FUNCTION_BLOCK FB_Transport_A
VAR_INPUT
	bStop1 :BOOL;
	bStop2 :BOOL;
	bStop3 :BOOL;
END_VAR
VAR_OUTPUT
	//Hardware Outputs
	bStopper1 :BOOL;
	bStopper2 :BOOL;
	bStopper3 :BOOL;
END_VAR
VAR
END_VAR

bStopper1 :=  bStop1;
bStopper2 :=  bStop2;
bStopper3 :=  bStop3;

END_FUNCTION_BLOCK

(* stored: Version 1.1.0.1
   POU FB_Transport_A: Id {6465c2c0-ecc4-47fa-9a2b-0303cbc4345b}, SpecialFunc None *)
